(* PLC project Generated.project, CODESYS CODESYS V3.5 SP19 Patch 1 *)
(* stored: creationDateTime 2026-09-06T13:00:42.447405, modificationDateTime 2026-09-06T13:00:42.447405 *)

(* ======================================================================= ⚖️ ST_fbWinch_Symmetry_Cfg — Configuration des seuils de symétrie M1/M2 ─────────────────────────────────────────────────────────────── 🎯 Rôle : Seuils de tolérance pour le diagnostic passif de symétrie treuils 📄 Doc métier : DOC/AF/AF_Partie-10_Fonction_Winch_v2.1.md ======================================================================= *)
TYPE ST_fbWinch_Symmetry_Cfg : STRUCT
  DeltaStartDelay_Ms : UDINT := 100;  (* Ecart max tolere au demarrage (ms) *)
  DeltaBrakeReleaseTime_Ms : UDINT := 100;  (* Ecart max temps desserrage frein (ms) *)
  DeltaBrakeApplyTime_Ms : UDINT := 100;  (* Ecart max temps serrage frein (ms) *)
  DeltaStopDistance_Mm : UDINT := 100;  (* Ecart max distance d'arret (mm) *)
  DeltaStopTime_Ms : UDINT := 200;  (* Ecart max temps d'arret (ms) *)
  MinimumCommandTime_Ms : UDINT := 1000;  (* Duree minimale de commande pour qualification (ms) *)
  MinimumSpeed_Mps : REAL := 0.05;  (* Vitesse minimale pour qualification (m/s) *)
END_STRUCT;
END_TYPE
